FUNCTION_BLOCK FB_SlaveArm
VAR_INPUT
END_VAR
VAR_OUTPUT
END_VAR
VAR
	// arm index, from 1 to 4
	m_armIdx: INT;
	
	// joints
	m_joints :ARRAY[1..g_sJntNum] OF FB_SlaveJoint;
	
	//  panel and insturment detect
	m_panelInstrumentOnIO AT%I*	:UDINT;
	m_panelDetect :FB_PanelDetect;
	m_instruDetect :FB_InstrumentDetect;
	m_instruNearDetect :FB_InstruNearDetect;
	m_panelOnFlag :BOOL:=FALSE;
	m_instruOnFlag :BOOL:=FALSE;
	m_instruNearFlag :BOOL:=FALSE;

	
	// trocar and  adjust detect
	m_adjustIO AT%I* :UDINT;
	m_adjustDetect :FB_AdjustDetect;
	m_trocarDetect : FB_TrocarDetect;
	m_adjustOnFlag :BOOL;
	m_trocarOnFlag :BOOL :=FALSE;
	m_adjustFallEdge :BOOL:=false;
	m_adjustFallEdgeDetect : F_TRIG;
	
	//endoscope type and posture switch
	m_endoscopeTypeSwitch : FB_IOToggleCheck;
	m_endoscopePostureSwitch : FB_IOToggleCheck;
	
	// instrument instance
	m_instrument : FB_Instrument;
	
	// instrument invasion depth before it's unmounted
	m_instruInvasionDepth :LREAL;

	// arm cartesian data, defined in each arm origin
	m_curCartPose	:ST_Frame;
	m_curCartTwist: Vec6d;
	m_cmdCartTwist :Vec6d;
	m_cmdCartPose:ST_Frame;
	
	// arm joint data
	m_curMotorPos :Vec8d;
	m_curLinkPos :Vec8d;
	m_curLinkSingle :Vec8d;
	m_curJntPos :Vec8d;
	m_curDHJntPos :Vec6d;
	m_curGripAngle :LREAL;
	m_curJntVel :Vec8d;
	m_curDHJntVel :Vec6d;
	m_curJntTrq :Vec8d;
	m_rawJntCurrent :Vec8d;
	m_filtJntCurrent :Vec8d;
	m_cmdJntTrq :Vec8d;
	m_cmdJntCurrent : Vec8d;
	m_cmdJntPos :Vec8d;
	m_cmdJntVel :Vec8d;
	
	// intrument joint backlash
	m_instruJntBacklash :Vec5d:=g_zeroVec5d;
		
	// arm dynamic data
	m_jntGravity : Vec8d:=g_zeroVec8d;
	m_jntMassMat : Mat3d;
	
	// arm jacobian and inverse
	m_jaco : Mat6d;
	
	// simulated status
	m_simJntPos :Vec8d;
	m_simDHJntPos :Vec6d;
	m_simGripAngle :LREAL;
	m_simCartPose : ST_Frame;
	m_simJaco : Mat6d;
	m_simJacoInv :Mat6d;
	m_isSingularity:BOOL:=false;
	
	// joint position controller
	m_jntPIDCtrl :ARRAY[1..g_sJntNum] OF FB_PID;
	
	// rising edge generator for instrument information reading
	m_ReadLDP:R_TRIG;
	
	// code execute time measure
	m_codeTime : Profiler;
	
END_VAR

PROPERTY adjustFallEdge : BOOL
GET
adjustFallEdge := m_adjustFallEdge;
END_GET
END_PROPERTY

PROPERTY adjustOn : bool
GET
adjustOn := m_adjustOnFlag;
END_GET
END_PROPERTY

PROPERTY armIdx : int
GET
armIdx:=m_armIdx;
END_GET
END_PROPERTY

METHOD PROTECTED calcJaco : BOOL
VAR_IN_OUT CONSTANT
	i_DHJntPos :Vec6d;
END_VAR
VAR_IN_OUT
	r_jaco :Mat6d;
END_VAR
VAR_INPUT
END_VAR

VAR
	d1, L, a, b :LREAL;
	q3:LREAL;

	c1,c2,c4,c5,c6,c7 :LREAL;
	s1,s2,s4,s5,s6,s7 :LREAL;

END_VAR
d1:=GVL_SlaveArmKinematic.g_d1;
L:=m_instrument.instruTypeInfo.m_rodLength;
a:=m_instrument.instruTypeInfo.m_headLength;
//b:=m_instrument.instruTypeInfo.m_fingerLength;
b:=0;

q3:=i_DHJntPos[3];
c1:=COS(i_DHJntPos[1]);
c2:=COS(i_DHJntPos[2]);
c4:=COS(i_DHJntPos[4]);
c5:=COS(i_DHJntPos[5]);
c6:=COS(i_DHJntPos[6]);

s1:=SIN(i_DHJntPos[1]);
s2:=SIN(i_DHJntPos[2]);
s4:=SIN(i_DHJntPos[4]);
s5:=SIN(i_DHJntPos[5]);
s6:=SIN(i_DHJntPos[6]);

// jacobian with DH joints
r_jaco[1,1]:=b*(c6*(c5*(c1*s4 - c2*c4*s1) + s1*s2*s5) - s6*(c1*c4 + c2*s1*s4)) + a*(c5*(c1*s4 - c2*c4*s1) + s1*s2*s5) - L*s1*s2 + q3*s1*s2;
r_jaco[1,2]:=-c1*(a*(c2*s5 + c4*c5*s2) - L*c2 + q3*c2 + b*(c6*(c2*s5 + c4*c5*s2) + s2*s4*s6));
r_jaco[1,3]:=-c1*s2;
r_jaco[1,4]:=s1*s2*(a*(c2*s5 + c4*c5*s2) + b*(c6*(c2*s5 + c4*c5*s2) + s2*s4*s6)) - c2*(b*(c6*(c5*(c1*s4 - c2*c4*s1) + s1*s2*s5) - s6*(c1*c4 + c2*s1*s4)) + a*(c5*(c1*s4 - c2*c4*s1) + s1*s2*s5));
r_jaco[1,5]:=- (a*(c2*s5 + c4*c5*s2) + b*(c6*(c2*s5 + c4*c5*s2) + s2*s4*s6))*(c1*c4 + c2*s1*s4) - s2*s4*(b*(c6*(c5*(c1*s4 - c2*c4*s1) + s1*s2*s5) - s6*(c1*c4 + c2*s1*s4)) + a*(c5*(c1*s4 - c2*c4*s1) + s1*s2*s5));
r_jaco[1,6]:= b*(c6*(c5*(c1*s4 - c2*c4*s1) + s1*s2*s5) - s6*(c1*c4 + c2*s1*s4))*(c2*c5 - c4*s2*s5) + b*(s5*(c1*s4 - c2*c4*s1) - c5*s1*s2)*(c6*(c2*s5 + c4*c5*s2) + s2*s4*s6);


r_jaco[2,1]:=0;
r_jaco[2,2]:=c1*(a*(c5*(s1*s4 + c1*c2*c4) - c1*s2*s5) + b*(c6*(c5*(s1*s4 + c1*c2*c4) - c1*s2*s5) - s6*(c4*s1 - c1*c2*s4)) + L*c1*s2 - q3*c1*s2) - s1*(b*(c6*(c5*(c1*s4 - c2*c4*s1) + s1*s2*s5) - s6*(c1*c4 + c2*s1*s4)) + a*(c5*(c1*s4 - c2*c4*s1) + s1*s2*s5) - L*s1*s2 + q3*s1*s2);
r_jaco[2,3]:= c2;
r_jaco[2,4]:=- s1*s2*(a*(c5*(s1*s4 + c1*c2*c4) - c1*s2*s5) + b*(c6*(c5*(s1*s4 + c1*c2*c4) - c1*s2*s5) - s6*(c4*s1 - c1*c2*s4))) - c1*s2*(b*(c6*(c5*(c1*s4 - c2*c4*s1) + s1*s2*s5) - s6*(c1*c4 + c2*s1*s4)) + a*(c5*(c1*s4 - c2*c4*s1) + s1*s2*s5));
r_jaco[2,5]:=(a*(c5*(s1*s4 + c1*c2*c4) - c1*s2*s5) + b*(c6*(c5*(s1*s4 + c1*c2*c4) - c1*s2*s5) - s6*(c4*s1 - c1*c2*s4)))*(c1*c4 + c2*s1*s4) - (b*(c6*(c5*(c1*s4 - c2*c4*s1) + s1*s2*s5) - s6*(c1*c4 + c2*s1*s4)) + a*(c5*(c1*s4 - c2*c4*s1) + s1*s2*s5))*(c4*s1 - c1*c2*s4);
r_jaco[2,6]:=b*(c6*(c5*(c1*s4 - c2*c4*s1) + s1*s2*s5) - s6*(c1*c4 + c2*s1*s4))*(s5*(s1*s4 + c1*c2*c4) + c1*c5*s2) - b*(s5*(c1*s4 - c2*c4*s1) - c5*s1*s2)*(c6*(c5*(s1*s4 + c1*c2*c4) - c1*s2*s5) - s6*(c4*s1 - c1*c2*s4));

r_jaco[3,1]:=a*(c5*(s1*s4 + c1*c2*c4) - c1*s2*s5) + b*(c6*(c5*(s1*s4 + c1*c2*c4) - c1*s2*s5) - s6*(c4*s1 - c1*c2*s4)) + L*c1*s2 - q3*c1*s2;
r_jaco[3,2]:=-s1*(a*(c2*s5 + c4*c5*s2) - L*c2 + q3*c2 + b*(c6*(c2*s5 + c4*c5*s2) + s2*s4*s6));
r_jaco[3,3]:=-s1*s2;
r_jaco[3,4]:=- c2*(a*(c5*(s1*s4 + c1*c2*c4) - c1*s2*s5) + b*(c6*(c5*(s1*s4 + c1*c2*c4) - c1*s2*s5) - s6*(c4*s1 - c1*c2*s4))) - c1*s2*(a*(c2*s5 + c4*c5*s2) + b*(c6*(c2*s5 + c4*c5*s2) + s2*s4*s6));
r_jaco[3,5]:=- (a*(c2*s5 + c4*c5*s2) + b*(c6*(c2*s5 + c4*c5*s2) + s2*s4*s6))*(c4*s1 - c1*c2*s4) - s2*s4*(a*(c5*(s1*s4 + c1*c2*c4) - c1*s2*s5) + b*(c6*(c5*(s1*s4 + c1*c2*c4) - c1*s2*s5) - s6*(c4*s1 - c1*c2*s4)));
r_jaco[3,6]:=b*(c6*(c5*(s1*s4 + c1*c2*c4) - c1*s2*s5) - s6*(c4*s1 - c1*c2*s4))*(c2*c5 - c4*s2*s5) + b*(c6*(c2*s5 + c4*c5*s2) + s2*s4*s6)*(s5*(s1*s4 + c1*c2*c4) + c1*c5*s2);

r_jaco[4,1]:=0;
r_jaco[4,2]:=-s1;
r_jaco[4,3]:=0;
r_jaco[4,4]:=-c1*s2;
r_jaco[4,5]:=c1*c2*s4 - c4*s1;
r_jaco[4,6]:=s5*(s1*s4 + c1*c2*c4) + c1*c5*s2;

r_jaco[5,1]:=-1;
r_jaco[5,2]:=0;
r_jaco[5,3]:=0;
r_jaco[5,4]:=c2;
r_jaco[5,5]:=s2*s4;
r_jaco[5,6]:=c4*s2*s5 - c2*c5;

r_jaco[6,1]:=0;
r_jaco[6,2]:=c1;
r_jaco[6,3]:=0;
r_jaco[6,4]:=-s1*s2;
r_jaco[6,5]:=c1*c4 + c2*s1*s4;
r_jaco[6,6]:=c5*s1*s2 - s5*(c1*s4 - c2*c4*s1);
END_METHOD

METHOD PROTECTED checkIO : BOOL
VAR_INPUT
END_VAR

VAR
	startFlag:BOOL;
END_VAR
// check adjust button
m_adjustOnFlag := m_adjustDetect.run(m_adjustIO);
m_adjustFallEdgeDetect(CLK:=m_adjustOnFlag, Q=>m_adjustFallEdge);

// check trocar
m_trocarOnFlag := m_trocarDetect.run(m_adjustIO);

// check panel and instrument
m_panelOnFlag := m_panelDetect.run(m_panelInstrumentOnIO);
m_instruOnFlag := m_instruDetect.run(m_panelInstrumentOnIO);
m_instruNearFlag := m_instruNearDetect.run(m_panelInstrumentOnIO);

//read instrument information
IF FALSE = m_instruOnFlag THEN
	m_instrument.reset();
END_IF
m_ReadLDP(CLK:= m_instruOnFlag, Q=>startFlag );
// try to read again if instrument ID is undefined
startFlag := startFlag OR m_instrument.onChipData.m_ErrorID = 1;
m_instrument.readParameters(startFlag);


// check endoscope type and posture 
// only check when electric Knife is off 
IF SlaveArmControl.m_masterRobotData.m_electricKnifePedalTrigger[1] = 0 AND SlaveArmControl.m_masterRobotData.m_electricKnifePedalTrigger[2] = 0 THEN
	IF m_endoscopeTypeSwitch.check((m_panelInstrumentOnIO AND 16#20)=32) THEN
		IF m_instrument.curScopeType = EndoScopeType_30 THEN
			m_instrument.nextScopeType := EndoscopeType_0;
		ELSE
			m_instrument.nextScopeType := EndoscopeType_30;
		END_IF
	END_IF
	IF m_endoscopePostureSwitch.check((m_panelInstrumentOnIO AND 16#10)=16) AND m_instrument.curScopeType = EndoScopeType_30  THEN
		IF m_instrument.curScopePosture = EndoScopePosture_HeadDown THEN
			m_instrument.nextScopePosture := EndoscopePosture_HeadUp;
		ELSE
			m_instrument.nextScopePosture := EndoScopePosture_HeadDown;
		END_IF
	END_IF
END_IF
END_METHOD

PROPERTY cmdCartPose : REFERENCE TO ST_Frame
GET
cmdCartPose REF= m_cmdCartPose;
END_GET
END_PROPERTY

PROPERTY cmdCartTwist : REFERENCE to Vec6d
GET
cmdCartTwist REF= m_cmdCartTwist;
END_GET
END_PROPERTY

PROPERTY cmdJntCurrent : REFERENCE TO  Vec8d
GET
cmdJntCurrent ref= m_cmdJntCurrent;
END_GET
END_PROPERTY

PROPERTY cmdJntPos : REFERENCE TO Vec8d
GET
cmdJntPos REF= m_cmdJntPos;
END_GET
END_PROPERTY

PROPERTY cmdJntTrq :REFERENCE TO Vec8d
GET
cmdJntTrq REF= m_cmdJntTrq;
END_GET
END_PROPERTY

PROPERTY cmdJntVel : REFERENCE TO Vec8d
GET
cmdJntVel REF= m_cmdJntVel;
END_GET
END_PROPERTY

PROPERTY curCartPose : REFERENCE TO ST_Frame
GET
curCartPose ref=m_curCartPose;
END_GET
END_PROPERTY

PROPERTY curCartTwist : REFERENCE TO Vec6d
GET
curCartTwist ref=m_curCartTwist;
END_GET
END_PROPERTY

PROPERTY curDHJntPos :REFERENCE TO Vec6d
GET
curDHJntPos ref= m_curDHJntPos;
END_GET
END_PROPERTY

PROPERTY curDHJntVel :REFERENCE TO Vec6d
GET
curDHJntVel REF= m_curDHJntVel;
END_GET
END_PROPERTY

PROPERTY curGripAngle : LREAL
GET
curGripAngle:=m_curGripAngle;
END_GET
END_PROPERTY

PROPERTY curJntPos : REFERENCE TO Vec8d
GET
curJntPos ref=m_curJntPos;
END_GET
END_PROPERTY

PROPERTY curJntTrq : REFERENCE TO Vec8d
GET
curJntTrq ref=m_curJntTrq;
END_GET
END_PROPERTY

PROPERTY curJntVel :REFERENCE TO Vec8d
GET
curJntVel ref=m_curJntVel;
END_GET
END_PROPERTY

PROPERTY curLinkPos :REFERENCE TO Vec8d
GET
curLinkPos ref=m_curLinkPos;
END_GET
END_PROPERTY

PROPERTY curMotorPos : REFERENCE TO  Vec8d
GET
curMotorPos ref=m_curMotorPos;
END_GET
END_PROPERTY

METHOD PUBLIC enable : BOOL
VAR_IN_OUT CONSTANT
	i_jntIdx :Vec8i;
END_VAR
VAR
	i :INT ;
END_VAR
FOR i:=1 TO g_sJntNum DO
	IF 1= i_jntIdx[i] THEN
		m_joints[i].enable();
	ELSE
		m_joints[i].disable();
	END_IF
END_FOR
END_METHOD

PROPERTY filtJntCurrent :REFERENCE TO Vec8d
GET
filtJntCurrent ref= m_filtJntCurrent;
END_GET
END_PROPERTY

// from active joint position to cartesian pose in arm origin
METHOD PROTECTED forwardKinematic : BOOL
VAR_IN_OUT CONSTANT
	i_DHJntPos :Vec6d;
END_VAR
VAR_IN_OUT
	r_cartPose :ST_Frame;
END_VAR
VAR
	d1, L, a, b :LREAL;
	q3 :LREAL;

	c1,c2,c4,c5,c6,c7 :LREAL;
	s1,s2,s4,s5,s6,s7 :LREAL;
	DHRot :Mat3d;
	
	tmpRot1,tmpRot2 : Mat3d;

END_VAR
d1:=GVL_SlaveArmKinematic.g_d1;
L:=m_instrument.instruTypeInfo.m_rodLength;
a:=m_instrument.instruTypeInfo.m_headLength;
//b:=m_instrument.instruTypeInfo.m_fingerLength;
b:=0;

q3:=i_DHJntPos[3];
c1:=COS(i_DHJntPos[1]);
c2:=COS(i_DHJntPos[2]);
c4:=COS(i_DHJntPos[4]);
c5:=COS(i_DHJntPos[5]);
c6:=COS(i_DHJntPos[6]);

s1:=SIN(i_DHJntPos[1]);
s2:=SIN(i_DHJntPos[2]);
s4:=SIN(i_DHJntPos[4]);
s5:=SIN(i_DHJntPos[5]);
s6:=SIN(i_DHJntPos[6]);


// cartesian pose frame
r_cartPose.m_pos[1]:=a*(c5*(s1*s4 + c1*c2*c4) - c1*s2*s5) + b*(c6*(c5*(s1*s4 + c1*c2*c4) - c1*s2*s5) - s6*(c4*s1 - c1*c2*s4)) + L*c1*s2 - q3*c1*s2;
r_cartPose.m_pos[2]:=a*(c2*s5 + c4*c5*s2) - d1 - L*c2 + q3*c2 + b*(c6*(c2*s5 + c4*c5*s2) + s2*s4*s6);
r_cartPose.m_pos[3]:=L*s1*s2 - a*(c5*(c1*s4 - c2*c4*s1) + s1*s2*s5) - b*(c6*(c5*(c1*s4 - c2*c4*s1) + s1*s2*s5) - s6*(c1*c4 + c2*s1*s4)) - q3*s1*s2;

DHRot[1,1]:= c6*(c5*(s1*s4 + c1*c2*c4) - c1*s2*s5) - s6*(c4*s1 - c1*c2*s4);
DHRot[2,1]:=c6*(c2*s5 + c4*c5*s2) + s2*s4*s6;
DHRot[3,1]:=s6*(c1*c4 + c2*s1*s4) - c6*(c5*(c1*s4 - c2*c4*s1) + s1*s2*s5);

DHRot[1,2]:=- s6*(c5*(s1*s4 + c1*c2*c4) - c1*s2*s5) - c6*(c4*s1 - c1*c2*s4);
DHRot[2,2]:=c6*s2*s4 - s6*(c2*s5 + c4*c5*s2);
DHRot[3,2]:=s6*(c5*(c1*s4 - c2*c4*s1) + s1*s2*s5) + c6*(c1*c4 + c2*s1*s4);

DHRot[1,3]:= s5*(s1*s4 + c1*c2*c4) + c1*c5*s2;
DHRot[2,3]:= c4*s2*s5 - c2*c5;
DHRot[3,3]:=c5*s1*s2 - s5*(c1*s4 - c2*c4*s1);

// convert to tcp rotation
matMultiply(DHRot, GVL_SlaveArmKinematic.g_tcpRotation, r_cartPOSE.m_rot);

//TODO: need verify
// rotate tcp coordinate 180 degree about z axis if instrument is a head-up 30deg endoscope
IF m_instrument.instruType = InstruType_Endoscope AND m_instrument.curScopeType = EndoScopeType_30 AND m_instrument.curScopePosture = EndoscopePosture_HeadUp THEN
	tmpRot2 := rotZ(pi);
	tmpRot1 := r_cartPOSE.m_rot;
	matMultiply(tmpRot1, tmpRot2, r_cartPOSE.m_rot);
END_IF
END_METHOD

METHOD PUBLIC init : BOOL
VAR_INPUT
	i_armIdx:INT;
END_VAR
VAR 
	i :INT ;
	currentRatioMotor2Jnt: LREAL;
END_VAR
// arm statues init
m_armIdx:=i_armIdx;
m_curGripAngle:=0;
m_simGripAngle:=0;
m_instruJntBacklash := g_zeroVec5d;

// joint init
FOR i:=1 TO g_sJntNum DO
	IF i<4 THEN
		m_joints[i].init(m_armIdx, i,g_slaveArmCtrlCycleTime, 1);
	ELSE
		m_joints[i].init(m_armIdx, i,g_slaveArmCtrlCycleTime, 4);
	END_IF
END_FOR

// init joint encoder and position calculation
initJntPos();

// joint controller init
FOR i:=1 TO g_sJntNum DO 
	currentRatioMotor2Jnt:=GVL_SlaveMotorParameters.g_motorTrqConst[i]*GVL_SlaveMotorParameters.g_motorReduction[i]/1000;
	m_jntPIDCtrl[i].init(g_slaveArmCtrlCycleTime,GVL_slaveControlParameters.g_posKp[i],GVL_slaveControlParameters.g_posKd[i],
		GVL_slaveControlParameters.g_posKi[i], GVL_slaveControlParameters.g_posKiLimit[i]* currentRatioMotor2Jnt,
		GVL_slaveControlParameters.g_posCtrlLimit[i]*currentRatioMotor2Jnt);
END_FOR

// instrument init
m_instrument.init(i_armIdx);

// endosocpe toggle button check
m_endoscopeTypeSwitch.init(0, 500);
m_endoscopePostureSwitch.init(0,500);
END_METHOD

METHOD PUBLIC initJntPos : BOOL
VAR_INPUT
END_VAR
VAR
	i:INT ;
END_VAR
// joint init
FOR i:=1 TO g_sJntNum DO
	m_joints[i].initJntPos();
END_FOR

// update arm status if joint position is re-init
updateStatus();
END_METHOD

PROPERTY instruJntBacklash :REFERENCE TO Vec5d
GET
instruJntBacklash ref=m_instruJntBacklash;
END_GET
SET
m_instruJntBacklash := instruJntBacklash;
END_SET
END_PROPERTY

PROPERTY instrument : REFERENCE TO FB_Instrument
GET
instrument REF=m_instrument;
END_GET
END_PROPERTY

PROPERTY instruNear : BOOL
GET
instruNear := m_instruNearFlag;
END_GET
END_PROPERTY

PROPERTY instruOn : bool
GET
instruOn:=m_instruOnFlag;
END_GET
END_PROPERTY

// check if instrument is in ready position(far enough from romote center) for following manipulation
METHOD PUBLIC instruReady : BOOL
VAR_INPUT
END_VAR

VAR
	// check buffer
	checkBuffer :LREAL := 0.005;
END_VAR
IF NOT(m_instrument.onChipData.m_InstruReadSucceed) THEN
	instruReady :=FALSE;
	RETURN;
END_IF

instruReady := m_curJntPos[3] < (m_instrument.instruTypeInfo.m_rodLength+m_instrument.instruTypeInfo.m_headLength
									+ m_instrument.instruTypeInfo.m_fingerLength - GVL_SlaveArmKinematic.g_minInstruRCDis+checkBuffer);
END_METHOD

METHOD PUBLIC isEnabled : BOOL
VAR_IN_OUT CONSTANT
	i_jntIdx :Vec8i;
END_VAR
VAR
	i :INT ;
END_VAR
isEnabled := TRUE;
FOR i:=1 TO g_sJntNum DO
	IF 1= i_jntIdx[i] THEN
		isEnabled :=  (m_joints[i].isEnabled() AND isEnabled);
	END_IF
END_FOR
END_METHOD

PROPERTY isSingurality : bool
GET
isSingurality:=m_isSingularity;
END_GET
END_PROPERTY

PROPERTY jaco :REFERENCE TO Mat6d
GET
jaco ref= m_jaco;
END_GET
END_PROPERTY

PROPERTY jntGravity :REFERENCE TO Vec8d
GET
jntGravity ref=m_jntGravity;
END_GET
END_PROPERTY

PROPERTY linkSingle : REFERENCE TO Vec8d
GET
linkSingle ref=m_curLinkSingle;
END_GET
END_PROPERTY

PROPERTY PUBLIC massMat :REFERENCE TO Mat3d
GET
massMat ref=m_jntMassMat;
END_GET
END_PROPERTY

METHOD PROTECTED modifyJaco : BOOL
VAR_IN_OUT CONSTANT
	i_DHJntPos :Vec6d;
END_VAR
VAR_IN_OUT
	r_jaco :Mat6d;
END_VAR

VAR CONSTANT
	// modify joint2/3 position to avoid jacobian singularity
	m_Jnt2PosThres :LREAL := -165 * g_deg2Rad;
	m_Jnt3PosThres :LREAL := -0.03;
END_VAR

VAR
	d1, L, a, b :LREAL;
	q2, q3:LREAL;

	c1,c2,c4,c5,c6,c7 :LREAL;
	s1,s2,s4,s5,s6,s7 :LREAL;
END_VAR
d1:=GVL_SlaveArmKinematic.g_d1;
L:=m_instrument.instruTypeInfo.m_rodLength;
a:=m_instrument.instruTypeInfo.m_headLength;
//b:=m_instrument.instruTypeInfo.m_fingerLength;
b:=0;

q2 := i_DHJntPos[2];
IF q2 < m_Jnt2PosThres THEN
	q2 := m_Jnt2PosThres;
END_IF

q3:=i_DHJntPos[3];
IF q3 - L > m_Jnt3PosThres THEN
	q3:= L + m_Jnt3PosThres;
END_IF

c1:=COS(i_DHJntPos[1]);
c2:=COS(q2);
c4:=COS(i_DHJntPos[4]);
c5:=COS(i_DHJntPos[5]);
c6:=COS(i_DHJntPos[6]);

s1:=SIN(i_DHJntPos[1]);
s2:=SIN(q2);
s4:=SIN(i_DHJntPos[4]);
s5:=SIN(i_DHJntPos[5]);
s6:=SIN(i_DHJntPos[6]);

// jacobian with DH joints
r_jaco[1,1]:=b*(c6*(c5*(c1*s4 - c2*c4*s1) + s1*s2*s5) - s6*(c1*c4 + c2*s1*s4)) + a*(c5*(c1*s4 - c2*c4*s1) + s1*s2*s5) - L*s1*s2 + q3*s1*s2;
r_jaco[1,2]:=-c1*(a*(c2*s5 + c4*c5*s2) - L*c2 + q3*c2 + b*(c6*(c2*s5 + c4*c5*s2) + s2*s4*s6));
r_jaco[1,3]:=-c1*s2;
r_jaco[1,4]:=s1*s2*(a*(c2*s5 + c4*c5*s2) + b*(c6*(c2*s5 + c4*c5*s2) + s2*s4*s6)) - c2*(b*(c6*(c5*(c1*s4 - c2*c4*s1) + s1*s2*s5) - s6*(c1*c4 + c2*s1*s4)) + a*(c5*(c1*s4 - c2*c4*s1) + s1*s2*s5));
r_jaco[1,5]:=- (a*(c2*s5 + c4*c5*s2) + b*(c6*(c2*s5 + c4*c5*s2) + s2*s4*s6))*(c1*c4 + c2*s1*s4) - s2*s4*(b*(c6*(c5*(c1*s4 - c2*c4*s1) + s1*s2*s5) - s6*(c1*c4 + c2*s1*s4)) + a*(c5*(c1*s4 - c2*c4*s1) + s1*s2*s5));
r_jaco[1,6]:= b*(c6*(c5*(c1*s4 - c2*c4*s1) + s1*s2*s5) - s6*(c1*c4 + c2*s1*s4))*(c2*c5 - c4*s2*s5) + b*(s5*(c1*s4 - c2*c4*s1) - c5*s1*s2)*(c6*(c2*s5 + c4*c5*s2) + s2*s4*s6);


r_jaco[2,1]:=0;
r_jaco[2,2]:=c1*(a*(c5*(s1*s4 + c1*c2*c4) - c1*s2*s5) + b*(c6*(c5*(s1*s4 + c1*c2*c4) - c1*s2*s5) - s6*(c4*s1 - c1*c2*s4)) + L*c1*s2 - q3*c1*s2) - s1*(b*(c6*(c5*(c1*s4 - c2*c4*s1) + s1*s2*s5) - s6*(c1*c4 + c2*s1*s4)) + a*(c5*(c1*s4 - c2*c4*s1) + s1*s2*s5) - L*s1*s2 + q3*s1*s2);
r_jaco[2,3]:= c2;
r_jaco[2,4]:=- s1*s2*(a*(c5*(s1*s4 + c1*c2*c4) - c1*s2*s5) + b*(c6*(c5*(s1*s4 + c1*c2*c4) - c1*s2*s5) - s6*(c4*s1 - c1*c2*s4))) - c1*s2*(b*(c6*(c5*(c1*s4 - c2*c4*s1) + s1*s2*s5) - s6*(c1*c4 + c2*s1*s4)) + a*(c5*(c1*s4 - c2*c4*s1) + s1*s2*s5));
r_jaco[2,5]:=(a*(c5*(s1*s4 + c1*c2*c4) - c1*s2*s5) + b*(c6*(c5*(s1*s4 + c1*c2*c4) - c1*s2*s5) - s6*(c4*s1 - c1*c2*s4)))*(c1*c4 + c2*s1*s4) - (b*(c6*(c5*(c1*s4 - c2*c4*s1) + s1*s2*s5) - s6*(c1*c4 + c2*s1*s4)) + a*(c5*(c1*s4 - c2*c4*s1) + s1*s2*s5))*(c4*s1 - c1*c2*s4);
r_jaco[2,6]:=b*(c6*(c5*(c1*s4 - c2*c4*s1) + s1*s2*s5) - s6*(c1*c4 + c2*s1*s4))*(s5*(s1*s4 + c1*c2*c4) + c1*c5*s2) - b*(s5*(c1*s4 - c2*c4*s1) - c5*s1*s2)*(c6*(c5*(s1*s4 + c1*c2*c4) - c1*s2*s5) - s6*(c4*s1 - c1*c2*s4));

r_jaco[3,1]:=a*(c5*(s1*s4 + c1*c2*c4) - c1*s2*s5) + b*(c6*(c5*(s1*s4 + c1*c2*c4) - c1*s2*s5) - s6*(c4*s1 - c1*c2*s4)) + L*c1*s2 - q3*c1*s2;
r_jaco[3,2]:=-s1*(a*(c2*s5 + c4*c5*s2) - L*c2 + q3*c2 + b*(c6*(c2*s5 + c4*c5*s2) + s2*s4*s6));
r_jaco[3,3]:=-s1*s2;
r_jaco[3,4]:=- c2*(a*(c5*(s1*s4 + c1*c2*c4) - c1*s2*s5) + b*(c6*(c5*(s1*s4 + c1*c2*c4) - c1*s2*s5) - s6*(c4*s1 - c1*c2*s4))) - c1*s2*(a*(c2*s5 + c4*c5*s2) + b*(c6*(c2*s5 + c4*c5*s2) + s2*s4*s6));
r_jaco[3,5]:=- (a*(c2*s5 + c4*c5*s2) + b*(c6*(c2*s5 + c4*c5*s2) + s2*s4*s6))*(c4*s1 - c1*c2*s4) - s2*s4*(a*(c5*(s1*s4 + c1*c2*c4) - c1*s2*s5) + b*(c6*(c5*(s1*s4 + c1*c2*c4) - c1*s2*s5) - s6*(c4*s1 - c1*c2*s4)));
r_jaco[3,6]:=b*(c6*(c5*(s1*s4 + c1*c2*c4) - c1*s2*s5) - s6*(c4*s1 - c1*c2*s4))*(c2*c5 - c4*s2*s5) + b*(c6*(c2*s5 + c4*c5*s2) + s2*s4*s6)*(s5*(s1*s4 + c1*c2*c4) + c1*c5*s2);

r_jaco[4,1]:=0;
r_jaco[4,2]:=-s1;
r_jaco[4,3]:=0;
r_jaco[4,4]:=-c1*s2;
r_jaco[4,5]:=c1*c2*s4 - c4*s1;
r_jaco[4,6]:=s5*(s1*s4 + c1*c2*c4) + c1*c5*s2;

r_jaco[5,1]:=-1;
r_jaco[5,2]:=0;
r_jaco[5,3]:=0;
r_jaco[5,4]:=c2;
r_jaco[5,5]:=s2*s4;
r_jaco[5,6]:=c4*s2*s5 - c2*c5;

r_jaco[6,1]:=0;
r_jaco[6,2]:=c1;
r_jaco[6,3]:=0;
r_jaco[6,4]:=-s1*s2;
r_jaco[6,5]:=c1*c4 + c2*s1*s4;
r_jaco[6,6]:=c5*s1*s2 - s5*(c1*s4 - c2*c4*s1);
END_METHOD

PROPERTY panelOn : bool
GET
panelOn :=m_panelOnFlag;
END_GET
END_PROPERTY

PROPERTY rawJntCurrent :REFERENCE TO Vec8d
GET
rawJntCurrent ref=m_rawJntCurrent;
END_GET
END_PROPERTY

// check if instrument is in ready position(far enough from romote center) for following manipulation
METHOD PUBLIC readyForInstruMount : BOOL
VAR_INPUT
END_VAR

VAR
	// check buffer
	checkBuffer :LREAL := 0.01;
	i:INT;
END_VAR
readyForInstruMount := (m_curJntPos[3]> GVL_SlaveMotorParameters.g_maxDHJntPos[3]-checkBuffer AND m_panelOnFlag);

// make sure instrument joint at zero position
FOR i:=4 TO 8 DO
	IF m_curLinkSingle[i]>1*g_deg2rad AND m_curLinkSingle[i]< g_2pi - 1*g_deg2rad THEN
		readyForInstruMount:=FALSE;
		EXIT;
	END_IF
END_FOR
END_METHOD

METHOD PUBLIC resetInstruDepth : BOOL
VAR_INPUT
END_VAR
m_instruInvasionDepth :=GVL_SlaveMotorParameters.g_maxJntPos[3];
END_METHOD

METHOD PUBLIC setInstruDepth : BOOL
VAR_INPUT
END_VAR
m_instruInvasionDepth := m_curJntPos[3]-m_instrument.instruTypeInfo.m_rodLength -
			COS(m_curDHJntPos[5]+pi/2) *( m_instrument.instruTypeInfo.m_headLength + m_instrument.instruTypeInfo.m_fingerLength * COS(m_curDHJntPos[6]));
END_METHOD

PROPERTY simCartPose :REFERENCE TO ST_Frame
GET
simCartPose ref=m_simCartPose;
END_GET
END_PROPERTY

PROPERTY simDHJntPos :REFERENCE TO Vec6d
GET
simDHJntPos ref= m_simDHJntPos;
END_GET
END_PROPERTY

PROPERTY simGripAngle : LREAL
GET
simGripAngle:=m_simGripAngle;
END_GET
END_PROPERTY

PROPERTY simJaco :REFERENCE TO mat6d
GET
simJaco ref=m_simJaco;
END_GET
END_PROPERTY

PROPERTY simJacoInv :REFERENCE TO Mat6d
GET
simJacoInv ref= m_simJacoInv;
END_GET
END_PROPERTY

PROPERTY PUBLIC trocarOn : bool
GET
trocarOn := m_trocarOnFlag;
END_GET
END_PROPERTY

// update joints control command
METHOD PUBLIC updateCmds : BOOL
VAR_IN_OUT CONSTANT
	i_armCtrlCmd : ST_SlaveArmCtrlCmds;
END_VAR
VAR
	i:INT;
END_VAR
m_cmdJntTrq:=i_armCtrlCmd.m_cmdJntTrq;
m_cmdJntPos :=i_armCtrlCmd.m_cmdJntPos;
m_cmdJntVel :=i_armCtrlCmd.m_cmdJntVel;
m_cmdCartTwist := i_armCtrlCmd.m_cmdCartTwist;
m_cmdCartPose :=i_armCtrlCmd.m_cmdCartPose;
m_simJntPos:=i_armCtrlCmd.m_simJntPos;

// update simulated master arm
updateSimStatus();

// enable/disable joints
enable(i_armCtrlCmd.m_jntEnableFlag);

m_codeTime(START:=TRUE, RESET:=TRUE);
// position/torque control
FOR i:=1 TO g_sJntNum DO 
	IF i_armCtrlCmd.m_jntOPMode[i]=DriverOPMode_PosTrq THEN
		// position controller and gravity feedforward
		m_cmdJntTrq[i]:=m_jntPIDCtrl[i].run(m_cmdJntPos[i],m_curJntPos[i],m_cmdJntVel[i],m_curJntVel[i]);
		m_cmdJntTrq[i]:=m_cmdJntTrq[i]+m_jntGravity[i] + i_armCtrlCmd.m_FFJntTrq[i];
		m_joints[i].updateCmds(DriverOPMode_Trq,m_cmdJntPos[i],m_cmdJntTrq[i]);
	ELSIF i_armCtrlCmd.m_jntOPMode[i]=DriverOPMode_Trq THEN
		// gravity feedforward
		m_jntPIDCtrl[i].reset();
		m_cmdJntTrq[i]:=m_cmdJntTrq[i]+m_jntGravity[i];
		m_joints[i].updateCmds(DriverOPMode_Trq,m_cmdJntPos[i],m_cmdJntTrq[i]);
	ELSE
		m_jntPIDCtrl[i].reset();
		m_cmdJntTrq[i]:=0;
		IF i>3 THEN
			// add instrument joint backlash
			m_joints[i].updateCmds(DriverOPMode_Pos,m_cmdJntPos[i]+m_instruJntBacklash[i-3],m_cmdJntTrq[i]);
		ELSE
			m_joints[i].updateCmds(DriverOPMode_Pos,m_cmdJntPos[i],m_cmdJntTrq[i]);
		END_IF
	END_IF
	
END_FOR
m_codeTime(START:=FALSE);
END_METHOD

METHOD PUBLIC updateDyna : BOOL
VAR_IN_out constant
	slaveDynaData : ST_SlaveDynaData;
END_VAR
m_jntMassMat:=slaveDynaData.m_massMat[m_armIdx];
m_jntGravity[1]:=slaveDynaData.m_gravity[m_armIdx][1];
m_jntGravity[2]:=slaveDynaData.m_gravity[m_armIdx][2];
m_jntGravity[3]:=slaveDynaData.m_gravity[m_armIdx][3];
END_METHOD

METHOD PUBLIC updateSimStatus : BOOL
VAR_INPUT
END_VAR
// instrument kinematic
m_instrument.instruFK(m_simJntPos, m_simDHJntPos, m_simGripAngle);

// simulated cartesion pose 
forwardKinematic(m_simDHJntPos,m_simCartPose);

// simulated jacobian
modifyJaco(m_simDHJntPos,m_simJaco);
m_isSingularity:=NOT(invMat6(m_simJaco, m_simJacoInv));
END_METHOD

// update arm status, including kinematic and dynamic
METHOD PUBLIC updateStatus : BOOL
VAR_INPUT
END_VAR
VAR 
	i,j:INT;
END_VAR
// update joint data
FOR i:=1 TO g_sJntNum DO
	m_joints[i].updateStatus();
END_FOR

// check IO informantion
checkIO();

// get joint data
FOR i:=1 TO g_sJntNum DO
	// remove instrument joint backlash
	IF i>3 THEN
		m_curMotorPos[i]:=m_joints[i].motorPos - m_instruJntBacklash[i-3];
		m_curLinkPos[i]:=m_joints[i].linkPos - m_instruJntBacklash[i-3];
		m_curLinkSingle[i]:=m_joints[i].linkSingle - m_instruJntBacklash[i-3];
		m_curJntPos[i]:=m_joints[i].jntPos - m_instruJntBacklash[i-3];
	ELSE
		m_curMotorPos[i]:=m_joints[i].motorPos;
		m_curLinkPos[i]:=m_joints[i].linkPos;
		m_curLinkSingle[i]:=m_joints[i].linkSingle;
		m_curJntPos[i]:=m_joints[i].jntPos;
	END_IF
	m_curJntVel[i]:=m_joints[i].jntVel;
	m_curJntTrq[i]:=m_joints[i].jntTrq;
	m_rawJntCurrent[i]:=m_joints[i].rawCurrent;
	m_filtJntCurrent[i]:=m_joints[i].filtCurrent;
	m_cmdJntCurrent[i]:=m_joints[i].cmdCurrent;
END_FOR 

// instrument kinematic
m_instrument.instruFK(m_curJntPos, m_curDHJntPos, m_curGripAngle);

// cartesion pose
forwardKinematic(m_curDHJntPos,m_curCartPose);

// jacobian
calcJaco(m_curDHJntPos,m_jaco);

// DH joint velocity
m_instrument.instruJntVelFK(m_curJntVel, m_curDHJntVel);

// cartesian twist
matMultiVec(m_jaco, m_curDHJntVel, m_curCartTwist);
END_METHOD

END_FUNCTION_BLOCK

(* stored: Version 1.1.0.1, ProductVersion 3.1.4024.12
   POU FB_SlaveArm: Id {623926f8-06e2-46b6-bb1f-baa6bc16e9cb}, SpecialFunc None
   Folder property: Id {4aa1799c-1556-4bc1-a713-06f14faa00f1}
   Property adjustFallEdge: Id {892fbc5d-bccd-475a-836d-3ab99edcd203}
   Get Get: Id {e41aaa50-cc49-4924-aa5c-7939e5c2aefd}
   Property adjustOn: Id {afc98598-ed29-4176-9f45-d842c4ec164a}
   Get Get: Id {d84a6e3e-5b0e-406e-b7c3-ff6a74a84739}
   Property armIdx: Id {1bcadfc3-0a4f-4bee-a1a7-b6d4d3a1eb58}
   Get Get: Id {198387ec-2e24-42e6-b0c2-2f769705d46f}
   Method calcJaco: Id {1172e5e4-b7f2-4690-a821-6304414cea84}
   Method checkIO: Id {613633aa-f5bc-4224-95e6-e974a90f8e6a}
   Property cmdCartPose: Id {72bf034f-e694-478b-8fc6-77f6ebb37ccd}
   Get Get: Id {cf508e47-c40b-4af1-9748-e64ccbaeea52}
   Property cmdCartTwist: Id {db564f7b-db8f-4a3a-ba4b-526788bb30bd}
   Get Get: Id {8a565392-e659-4e2f-8d16-f053ffd74289}
   Property cmdJntCurrent: Id {cbd7aa84-e545-47b8-bdc5-960aa8409c91}
   Get Get: Id {12be56c2-8b79-47d6-b1f2-86b8e0a5f91a}
   Property cmdJntPos: Id {fe3eaf75-296c-46e0-a9c6-f78064c649e8}
   Get Get: Id {21440cc7-9bce-4ec3-adb3-863b046ec9da}
   Property cmdJntTrq: Id {a8b8f509-6313-4dea-add6-0d9f63644d17}
   Get Get: Id {69ae4f04-ab57-4161-852a-de73ff986ad6}
   Property cmdJntVel: Id {8b50ea35-c0ee-4521-ab63-6cd2fbfd419a}
   Get Get: Id {32d77105-7aae-4d69-88ee-4b488832fd1d}
   Property curCartPose: Id {d18be23c-99e5-435e-8688-90e0fb3be9ca}
   Get Get: Id {013b03f6-adb7-4855-b0fe-353f77f67094}
   Property curCartTwist: Id {e4b7010c-887c-41fa-8766-1a9192e9d06a}
   Get Get: Id {b7c89bf7-90fc-4841-be25-e467b1918b68}
   Property curDHJntPos: Id {a2be2c30-01e0-4901-99e6-385cb59adf34}
   Get Get: Id {5292b7b6-7cd6-4d1f-a863-39df8105a863}
   Property curDHJntVel: Id {e70b9eba-b60c-47ce-ba40-0d867f7d1681}
   Get Get: Id {f89a1342-80b1-4a57-8483-5c3af208683c}
   Property curGripAngle: Id {5187a911-df75-4b56-8b45-38142d9b24de}
   Get Get: Id {871729fd-1ba1-4906-aec3-7d572491feb2}
   Property curJntPos: Id {d72c054a-bae9-44cb-97ff-fe7c76c53cb8}
   Get Get: Id {332d5297-fb56-44bd-a751-714464e0813c}
   Property curJntTrq: Id {8c78ba58-302c-4844-9d36-e487700a0e19}
   Get Get: Id {1767bffb-cddd-4133-ad6f-5125f86340af}
   Property curJntVel: Id {904c68d5-30c9-4ed3-b3c5-6bcd345bcd5a}
   Get Get: Id {0a508621-c577-4d50-8cc3-bd8133f79f72}
   Property curLinkPos: Id {3725bf51-2c50-4574-b2a7-e2af9fd4da29}
   Get Get: Id {cff7c92f-5276-4a58-b7ca-f6248868b409}
   Property curMotorPos: Id {ad9d9e24-10f4-4dc4-b0d2-86517dead53b}
   Get Get: Id {bc557e46-3cdd-47ba-9e7f-cf7525f3969d}
   Method enable: Id {596f2892-08b6-4851-84d5-1537c558264e}
   Property filtJntCurrent: Id {1f5e4c97-ef8c-417a-90ec-656c048c0e4f}
   Get Get: Id {34ea0c3d-b0bc-4adb-bbb3-f4ab6640a7ff}
   Method forwardKinematic: Id {182b544f-f7c4-475e-8af7-8c07aa230234}
   Method init: Id {d7bcc040-c32e-4455-ab43-70de0dc2919e}
   Method initJntPos: Id {56ee4071-fcb1-4318-b1b9-837ea21e1627}
   Property instruJntBacklash: Id {88009436-63a3-453e-90cc-655a8a6c10d7}
   Get Get: Id {042c0ee1-c963-40d8-8b91-055199bc99cd}
   Set Set: Id {f4769db0-ca40-4b10-b4c1-f1e63de83403}
   Property instrument: Id {ef5d0758-d499-4e04-a177-87950f9a716b}
   Get Get: Id {3a5249de-ec45-4e88-a302-3df6650a3ff5}
   Property instruNear: Id {29bf66f9-822d-4749-92c9-ee092b53b459}
   Get Get: Id {6b30ea9b-f7b2-4aff-9934-1c8f2b6bc1de}
   Property instruOn: Id {4486d0c9-79b0-4e6c-acfb-23ca16ba44f5}
   Get Get: Id {daa69233-49df-439c-8476-605873205ebf}
   Method instruReady: Id {4f7fb741-1810-447d-a3ef-fca916ec7903}
   Method isEnabled: Id {00a67cf8-62b1-4004-a2ca-9469bb0f3cab}
   Property isSingurality: Id {da3c3ca8-d645-443c-af9d-86ff4ca01cff}
   Get Get: Id {69dc0611-36d4-4919-91ba-cfdefe53366b}
   Property jaco: Id {2c2ce445-b511-4254-9c8e-e5667e1b6bdb}
   Get Get: Id {27a6e900-c6e6-40c0-aa03-4dc0d1214554}
   Property jntGravity: Id {72dbb3a4-f37f-4edd-afb1-2190cd1f62fc}
   Get Get: Id {5c8a2ae5-eaad-400d-b638-ec46a75b5ccb}
   Property linkSingle: Id {23452807-9686-4e19-a62d-225c05ba29f3}
   Get Get: Id {f3f0fe9c-39ae-4e13-ac6a-e473233979ba}
   Property massMat: Id {c4fbf6a1-1d71-4f80-9bfa-395c19261a6f}
   Get Get: Id {b8079ba8-3835-474b-9d8e-6afd86dc6a9b}
   Method modifyJaco: Id {d0ec41d7-ce80-43b2-a117-9fcbd2b4368b}
   Property panelOn: Id {38ffa1da-012d-4dbc-ad5b-314577ed285b}
   Get Get: Id {b8c5f533-4196-44c4-9a48-01cc1ca3c250}
   Property rawJntCurrent: Id {f1221838-7bcd-4d84-b9f8-7dc96a864978}
   Get Get: Id {23a8503d-4e33-47db-b530-039bdd0d530f}
   Method readyForInstruMount: Id {70a1cabf-0568-4973-adb8-2d2bf84e7996}
   Method resetInstruDepth: Id {442cf664-eb0b-4d84-a453-ceda2815dd97}
   Method setInstruDepth: Id {f666f43c-697b-4bc4-8326-000cbf8a2e4d}
   Property simCartPose: Id {6426ffc4-f74f-4984-ac32-a9f9d8b8c8ca}
   Get Get: Id {a61bb7de-a7ad-4b34-8063-e53c825d0db4}
   Property simDHJntPos: Id {c6c26215-f204-4db3-9793-ef759045910e}
   Get Get: Id {52d60fe7-649d-4c54-a901-14c6c6eee89d}
   Property simGripAngle: Id {4ec8904f-ef0e-46d6-9b7d-280a45e21cf5}
   Get Get: Id {6dc37561-5d97-45fe-bee2-ebd740ec58ce}
   Property simJaco: Id {0fa24ffb-bfb3-496c-82de-08842f53e6e4}
   Get Get: Id {35c7dda2-112e-4042-99cd-4eac5d67ff5e}
   Property simJacoInv: Id {9bccb200-445a-4f96-a4eb-1e257b2cb058}
   Get Get: Id {2b6988d5-cc9a-4745-b2b4-b07fc10b1b71}
   Property trocarOn: Id {ad96c106-befc-48a9-abe7-5d7b42881f88}
   Get Get: Id {bb55ac1e-1079-48fa-ba1e-bc9844803f5a}
   Method updateCmds: Id {4f271d3a-4b2b-4f85-986e-f8fdffb5994c}
   Method updateDyna: Id {02de28e3-c8a7-46cf-834a-5bf048b5e039}
   Method updateSimStatus: Id {f15ad7c2-6655-4b50-9555-9aa968e8753f}
   Method updateStatus: Id {21b3fe9a-0eba-4313-bb9a-33b1f0038771} *)
